// TIA Portal V19 export
DATA_BLOCK "A0302_Bordatrice_RegolazioneFormato_PERS"   // DB71
// stored: MemoryReserve 100
   VAR RETAIN
      Par_Machine : Struct
         Nervatura_Pos_Riposo : Real := 2.0;
         Passaggio01_MaxDisallineamentoAXs : Real := 0.5;   // (Controllo disabilitato se <= 0)
         Passaggio02_MaxDisallineamentoAXs : Real := 0.5;   // (Controllo disabilitato se <= 0)
         Passaggio03_MaxDisallineamentoAXs : Real := 0.5;   // (Controllo disabilitato se <= 0)
         Passaggio04_MaxDisallineamentoAXs : Real := 0.5;   // (Controllo disabilitato se <= 0)
         AxD_AutoSpeed { ExternalAccessible := 'False'; ExternalVisible := 'False'; ExternalWritable := 'False'} : Real := 100.0;
      END_STRUCT;
      Par_Enc : Array[1..9] of "PosFbk_RTN";
      Par_D { S7_SetPoint := 'True'} : Array[1..1] of "Positioning_DOL_Machine_Par";
      Par_M : Array[2..9] of "Positioning_MOL_Machine_Par";
      Pers_D { S7_SetPoint := 'True'} : Array[1..1] of "Positioning_DOL_Machine_Pers_Data";
      Pers_M : Array[2..9] of "Positioning_MOL_Machine_Pers_Data";
   END_VAR
BEGIN
   Par_Enc[1].Preset.Pulses := -1_814_114_496;
   Par_Enc[2].Preset.Pulses := -2_062_495_152;
   Par_Enc[3].Preset.Pulses := -1_142_247_532;
   Par_Enc[4].Preset.Pulses := 1_928_214_608;
   Par_Enc[5].Preset.Pulses := -519_364_864;
   Par_Enc[6].Preset.Pulses := -1_662_099_024;
   Par_Enc[7].Preset.Pulses := -1_564_817_400;
   Par_Enc[8].Preset.Pulses := 754_806_652;
   Par_Enc[9].Preset.Pulses := 904_129_836;
   Par_Enc[1].Preset.Units := 180.0;
   Par_Enc[2..9].Preset.Units := 45.0;
   Par_Enc[1].Config.Resolution := -0.2;
   Par_Enc[2..9].Config.Resolution := -1.0;
   Par_D[1].PosTolerance := 0.1;
   Par_D[1].Minus_Limit := 59.0;
   Par_D[1].Plus_Limit := 215.0;
   Par_D[1].PreCutOff := 0.1;
   Par_D[1].PreEndLowSpeed := 1.0;
   Par_D[1].PreEndMedSpeed := 5.0;
   Par_D[1].LowSpeed := 35.0;
   Par_D[1].MedSpeed := 70.0;
   Par_D[1].HighSpeed := 70.0;
   Par_D[1].Man_Speed := 100.0;
   Par_M[2..9].PosTolerance := 0.1;
   Par_M[2..9].DelayInPosition := T#100MS;
   Par_M[2..8].Minus_Limit := 38.0;
   Par_M[9].Minus_Limit := 38.5;
   Par_M[2..9].Plus_Limit := 52.0;
   Par_M[2..9].PreCutOff := 0.03;
   Pers_D[1].AxisHomed := TRUE;
   Pers_M[2..9].AxisHomed := TRUE;
END_DATA_BLOCK
